FUNCTION_BLOCK FB_ControlReset_SC
VAR_INPUT
	fVelRef			: LREAL;
	ferror			: LREAL;

END_VAR
VAR_OUTPUT
	bReset			: BOOL;
END_VAR
VAR
	ferror_Tolerence	: LREAL := 0.001;
END_VAR

IF fVelRef = 0.0 AND ABS(ferror) < ferror_Tolerence THEN
	bReset := TRUE;
ELSE
	bReset := FALSE;
END_IF

END_FUNCTION_BLOCK

(* stored: Version 1.1.0.1
   POU FB_ControlReset_SC: Id {8003dd09-0a5a-4824-b0f6-9417fe90b905}, SpecialFunc None *)
